// TIA Portal V19 export
TYPE "LUC_typeSignalStackByDWord"
// Stack Light Signals by DWord
// stored: Access Published
   STRUCT
      statusByDWord { ExternalWritable := 'False'} : DWord;   // Stack light status. Indicates the current active lights and their behaviour.
   END_STRUCT;
END_TYPE
